{attribute 'GeneratedUsingTerminal: APS4322-7000-0017'}
{attribute addProperty BoxType "APS4322-7000-0017"}
{attribute addProperty Id "CommControlWordAT %Q*UINT2Data_1AT %Q*UINT2"}
{attribute addProperty CRC "136315556"}
{attribute addProperty Size "4"}
TYPE APS_Comm_Outputs_082002A4 :
STRUCT
	{attribute addProperty Name "CommControlWord"}
	CommControlWord AT %Q* : UINT;
	{attribute addProperty Name "Data_1"}
	Data_1 AT %Q* : UINT;
END_STRUCT
END_TYPE

(* stored: Version 1.2.0.0, ProductVersion 3.1.4024.9
   DUT APS_Comm_Outputs_082002A4: Id {c08cee31-8bce-4246-8a18-cc32d6b276d4} *)
